Fanuc TP program (LS listing): UP002.LS

/PROG  UP002
/ATTR
OWNER		= AUROM;
COMMENT		= "Soldadura Est.";
PROG_SIZE	= 20204;
CREATE		= DATE 23-02-08  TIME 21:26:18;
MODIFIED	= DATE 24-04-03  TIME 04:58:58;
FILE_NAME	= UP002;
VERSION		= 0;
LINE_COUNT	= 81;
MEMORY_SIZE	= 39340;
PROTECT		= READ_WRITE;
TCD:  STACK_SIZE	= 500,
      TASK_PRIORITY	= 50,
      TIME_SLICE	= 0,
      BUSY_LAMP_OFF	= 0,
      ABORT_REQUEST	= 0,
      PAUSE_REQUEST	= 0;
DEFAULT_GROUP	= 1,1,1,1,*;
CONTROL_CODE	= 00000001 00000000;
/APPL
/MN
   1:  UFRAME_NUM=1 ;
   2:  UTOOL_NUM=2 ;
   3:  PAYLOAD[2] ;
   4:J P[1] 100% CNT0 ACC100 TB    .10sec,P-SPS    ;
      1:  TC_ONLINE (ON) ;
      2:  DO[23]=OFF ;
      3:  TIMER[4]=RESET ;
      4:  TIMER[4]=START ;
      5:  CALL MAKRO050    ;
      6:  !Lib. de Herramientas ;
      7:  DO[80]=ON ;
      8:  DO[78]=OFF ;
      9:  DO[77]=ON ;
     10:  DO[75]=OFF ;
     11:  !Lib. de Anticolisiones ;
     12:  DO[45]=ON ;
     13:  DO[46]=ON ;
     14:  !Apagar Posicion Base ;
     15:  DO[15]=OFF ;
     16:  !Roboter auf der Bahn ;
     17:  DO[16]=ON ;
     18:  !Basculante 1 en Pos. de Reposo ;
     19:  IF (!DI[842] AND DO[12]),CALL MAKRO072 ;
     20:  WAIT (M[96])    ;
     21:  WAIT (DI[23])    ;
     22:  DO[23]=(ON) ;
     23:  TC_ONLINE (M[1] AND M[30] AND M[32] AND M[33] AND M[95] AND M[96]) ;
       ------ ;
   5:J P[2] 100% CNT100 ACC100 TB   0.00sec,P-SPS    ;
      1:  TC_ONLINE (M[1] AND M[30] AND M[32] AND M[33] AND M[95] AND M[96]) ;
       ------ ;
   6:J P[3] 100% CNT100 ACC100 TB   0.00sec,P-SPS    ;
      1:  TC_ONLINE (M[1] AND M[30] AND M[32] AND M[33] AND M[95] AND M[96]) ;
       ------ ;
   7:J P[4] 100% CNT100 ACC100 TB   0.00sec,P-SPS    ;
      1:  TC_ONLINE (M[1] AND M[30] AND M[32] AND M[33] AND M[95] AND M[96]) ;
       ------ ;
   8:J P[5] 100% CNT90 ACC80 TB   0.00sec,P-SPS    ;
      1:  TC_ONLINE (M[1] AND M[30] AND M[32] AND M[33] AND M[95] AND M[96]) ;
       ------ ;
   9:  !5QA802035_014_O_PS_0007 ;
  10:  !Punto de Sol. No. 5737 ;
  11:J P[6] 100% CNT10 ACC80 TB    .10sec,P-SPS Offset,PR[11]    ;
      1:  TC_ONLINE (ON) ;
      2:  DO[23]=OFF ;
      3:  WAIT (!DI[16] AND DI[23])    ;
      4:  CALL VW_USER(Basic1,EZSP,Nr1,ProgNr=99, , ,S-Punkt=5737,Fzg_Typ=3,EIN/AUS=ON) ;
      5:  GO[2]=(R[197]) ;
      6:  WAIT (!DI[129] OR DI[26])    ;
      7:  CALL MAKRO080    ;
      8:  WAIT (DI[23])    ;
      9:  DO[23]=ON ;
     10:  TC_ONLINE (M[1] AND M[30] AND M[32] AND M[33] AND M[95] AND M[96]) ;
       ------ ;
  12:  !5QA802035_014_O_PS_0008 ;
  13:  !Punto de Sol. No. 5738 ;
  14:J P[7] 100% CNT0 ACC100 TB    .10sec,P-SPS Offset,PR[11]    ;
      1:  TC_ONLINE (ON) ;
      2:  DO[23]=OFF ;
      3:  WAIT (!DI[16] AND DI[23])    ;
      4:  CALL VW_USER(Basic1,EZSP,Nr1,ProgNr=99, , ,S-Punkt=5738,Fzg_Typ=3,EIN/AUS=ON) ;
      5:  GO[2]=(R[197]) ;
      6:  WAIT (!DI[129] OR DI[26])    ;
      7:  CALL MAKRO080    ;
      8:  WAIT (DI[23])    ;
      9:  DO[23]=ON ;
     10:  TC_ONLINE (M[1] AND M[30] AND M[32] AND M[33] AND M[95] AND M[96]) ;
       ------ ;
  15:  !5QA802035_014_O_PS_0009 ;
  16:  !Punto de Sol. No. 5739 ;
  17:J P[8] 100% CNT0 ACC100 TB    .10sec,P-SPS Offset,PR[11]    ;
      1:  TC_ONLINE (ON) ;
      2:  DO[23]=OFF ;
      3:  WAIT (!DI[16] AND DI[23])    ;
      4:  CALL VW_USER(Basic1,EZSP,Nr1,ProgNr=99, , ,S-Punkt=5739,Fzg_Typ=3,EIN/AUS=ON) ;
      5:  GO[2]=(R[197]) ;
      6:  WAIT (!DI[129] OR DI[26])    ;
      7:  CALL MAKRO080    ;
      8:  WAIT (DI[23])    ;
      9:  DO[23]=ON ;
     10:  TC_ONLINE (M[1] AND M[30] AND M[32] AND M[33] AND M[95] AND M[96]) ;
       ------ ;
  18:  !5QA802035_030_AE_PS_0004 ;
  19:  !Punto de Sol. No. 5740 ;
  20:J P[9] 100% CNT0 ACC100 TB    .10sec,P-SPS Offset,PR[11]    ;
      1:  TC_ONLINE (ON) ;
      2:  DO[23]=OFF ;
      3:  WAIT (!DI[16] AND DI[23])    ;
      4:  CALL VW_USER(Basic1,EZSP,Nr1,ProgNr=99, , ,S-Punkt=5740,Fzg_Typ=3,EIN/AUS=ON) ;
      5:  GO[2]=(R[197]) ;
      6:  WAIT (!DI[129] OR DI[26])    ;
      7:  CALL MAKRO080    ;
      8:  WAIT (DI[23])    ;
      9:  DO[23]=ON ;
     10:  TC_ONLINE (M[1] AND M[30] AND M[32] AND M[33] AND M[95] AND M[96]) ;
       ------ ;
  21:  !5QA802035_030_AE_PS_0005 ;
  22:  !Punto de Sol. No. 5741 ;
  23:J P[10] 100% CNT0 ACC100 TB    .10sec,P-SPS Offset,PR[11]    ;
      1:  TC_ONLINE (ON) ;
      2:  DO[23]=OFF ;
      3:  WAIT (!DI[16] AND DI[23])    ;
      4:  CALL VW_USER(Basic1,EZSP,Nr1,ProgNr=99, , ,S-Punkt=5741,Fzg_Typ=3,EIN/AUS=ON) ;
      5:  GO[2]=(R[197]) ;
      6:  WAIT (!DI[129] OR DI[26])    ;
      7:  CALL MAKRO080    ;
      8:  WAIT (DI[23])    ;
      9:  DO[23]=ON ;
     10:  TC_ONLINE (M[1] AND M[30] AND M[32] AND M[33] AND M[95] AND M[96]) ;
       ------ ;
  24:J P[11] 100% CNT100 ACC100 TB   0.00sec,P-SPS    ;
      1:  TC_ONLINE (M[1] AND M[30] AND M[32] AND M[33] AND M[95] AND M[96]) ;
       ------ ;
  25:  !5QA802035_030_AE_PS_0006 ;
  26:  !Punto de Sol. No. 5742 ;
  27:J P[12] 100% CNT0 ACC100 TB    .10sec,P-SPS Offset,PR[11]    ;
      1:  TC_ONLINE (ON) ;
      2:  DO[23]=OFF ;
      3:  WAIT (!DI[16] AND DI[23])    ;
      4:  CALL VW_USER(Basic1,EZSP,Nr1,ProgNr=99, , ,S-Punkt=5742,Fzg_Typ=3,EIN/AUS=ON) ;
      5:  GO[2]=(R[197]) ;
      6:  WAIT (!DI[129] OR DI[26])    ;
      7:  CALL MAKRO080    ;
      8:  WAIT (DI[23])    ;
      9:  DO[23]=ON ;
     10:  TC_ONLINE (M[1] AND M[30] AND M[32] AND M[33] AND M[95] AND M[96]) ;
       ------ ;
  28:J P[13] 100% CNT100 ACC100 TB   0.00sec,P-SPS    ;
      1:  TC_ONLINE (M[1] AND M[30] AND M[32] AND M[33] AND M[95] AND M[96]) ;
       ------ ;
  29:J P[14] 100% CNT100 ACC100 TB    .10sec,P-SPS    ;
      1:  TC_ONLINE (M[1] AND M[30] AND M[32] AND M[33] AND M[95] AND M[96]) ;
       ------ ;
  30:  !5QA802035_034_AJ_PS_0001 ;
  31:  !Punto de Sol. No. 5743 ;
  32:J P[15] 100% CNT0 ACC100 TB    .10sec,P-SPS Offset,PR[11]    ;
      1:  TC_ONLINE (ON) ;
      2:  DO[23]=OFF ;
      3:  WAIT (!DI[16] AND DI[23])    ;
      4:  CALL VW_USER(Basic1,EZSP,Nr1,ProgNr=99, , ,S-Punkt=5743,Fzg_Typ=3,EIN/AUS=ON) ;
      5:  GO[2]=(R[197]) ;
      6:  WAIT (!DI[129] OR DI[26])    ;
      7:  CALL MAKRO080    ;
      8:  WAIT (DI[23])    ;
      9:  DO[23]=ON ;
     10:  TC_ONLINE (M[1] AND M[30] AND M[32] AND M[33] AND M[95] AND M[96]) ;
       ------ ;
  33:  !5QA802035_034_AJ_PS_0003 ;
  34:  !Punto de Sol. No. 5744 ;
  35:J P[16] 100% CNT0 ACC100 TB    .10sec,P-SPS Offset,PR[11]    ;
      1:  TC_ONLINE (ON) ;
      2:  DO[23]=OFF ;
      3:  WAIT (!DI[16] AND DI[23])    ;
      4:  CALL VW_USER(Basic1,EZSP,Nr1,ProgNr=99, , ,S-Punkt=5744,Fzg_Typ=3,EIN/AUS=ON) ;
      5:  GO[2]=(R[197]) ;
      6:  WAIT (!DI[129] OR DI[26])    ;
      7:  CALL MAKRO080    ;
      8:  WAIT (DI[23])    ;
      9:  DO[23]=ON ;
     10:  TC_ONLINE (M[1] AND M[30] AND M[32] AND M[33] AND M[95] AND M[96]) ;
       ------ ;
  36:J P[17] 100% CNT100 ACC100 TB   0.00sec,P-SPS    ;
      1:  TC_ONLINE (M[1] AND M[30] AND M[32] AND M[33] AND M[95] AND M[96]) ;
       ------ ;
  37:J P[18] 100% CNT100 ACC100 TB   0.00sec,P-SPS    ;
      1:  TC_ONLINE (M[1] AND M[30] AND M[32] AND M[33] AND M[95] AND M[96]) ;
       ------ ;
  38:  !5QA802035_048_BL_PS_0001 ;
  39:  !Punto de Sol. No. 5749 ;
  40:J P[19] 100% CNT0 ACC100 TB    .10sec,P-SPS Offset,PR[11]    ;
      1:  TC_ONLINE (ON) ;
      2:  DO[23]=OFF ;
      3:  WAIT (!DI[16] AND DI[23])    ;
      4:  CALL VW_USER(Basic1,EZSP,Nr1,ProgNr=99, , ,S-Punkt=5749,Fzg_Typ=3,EIN/AUS=ON) ;
      5:  GO[2]=(R[197]) ;
      6:  WAIT (!DI[129] OR DI[26])    ;
      7:  CALL MAKRO080    ;
      8:  WAIT (DI[23])    ;
      9:  DO[23]=ON ;
     10:  TC_ONLINE (M[1] AND M[30] AND M[32] AND M[33] AND M[95] AND M[96]) ;
       ------ ;
  41:J P[20] 100% CNT100 ACC100 TB   0.00sec,P-SPS    ;
      1:  TC_ONLINE (M[1] AND M[30] AND M[32] AND M[33] AND M[95] AND M[96]) ;
       ------ ;
  42:J P[21] 100% CNT100 ACC100 TB   0.00sec,P-SPS    ;
      1:  TC_ONLINE (M[1] AND M[30] AND M[32] AND M[33] AND M[95] AND M[96]) ;
       ------ ;
  43:J P[22] 100% CNT100 ACC100 TB   0.00sec,P-SPS    ;
      1:  TC_ONLINE (M[1] AND M[30] AND M[32] AND M[33] AND M[95] AND M[96]) ;
       ------ ;
  44:J P[23] 100% CNT100 ACC100 TB   0.00sec,P-SPS    ;
      1:  TC_ONLINE (M[1] AND M[30] AND M[32] AND M[33] AND M[95] AND M[96]) ;
       ------ ;
  45:J P[24] 100% CNT100 ACC100 TB   0.00sec,P-SPS    ;
      1:  TC_ONLINE (M[1] AND M[30] AND M[32] AND M[33] AND M[95] AND M[96]) ;
       ------ ;
  46:J P[25] 100% CNT100 ACC100 TB   0.00sec,P-SPS    ;
      1:  TC_ONLINE (M[1] AND M[30] AND M[32] AND M[33] AND M[95] AND M[96]) ;
       ------ ;
  47:J P[26] 100% CNT100 ACC100 TB   0.00sec,P-SPS    ;
      1:  TC_ONLINE (M[1] AND M[30] AND M[32] AND M[33] AND M[95] AND M[96]) ;
       ------ ;
  48:J P[27] 100% CNT100 ACC100 TB   0.00sec,P-SPS    ;
      1:  TC_ONLINE (M[1] AND M[30] AND M[32] AND M[33] AND M[95] AND M[96]) ;
       ------ ;
  49:J P[28] 100% CNT100 ACC100 TB   0.00sec,P-SPS    ;
      1:  TC_ONLINE (M[1] AND M[30] AND M[32] AND M[33] AND M[95] AND M[96]) ;
       ------ ;
  50:J P[29] 100% CNT100 ACC100 TB   0.00sec,P-SPS    ;
      1:  TC_ONLINE (M[1] AND M[30] AND M[32] AND M[33] AND M[95] AND M[96]) ;
       ------ ;
  51:J P[30] 100% CNT100 ACC100 TB   0.00sec,P-SPS    ;
      1:  TC_ONLINE (M[1] AND M[30] AND M[32] AND M[33] AND M[95] AND M[96]) ;
       ------ ;
  52:J P[31] 100% CNT100 ACC100 TB   0.00sec,P-SPS    ;
      1:  TC_ONLINE (M[1] AND M[30] AND M[32] AND M[33] AND M[95] AND M[96]) ;
       ------ ;
  53:J P[32] 100% CNT100 ACC100 TB   0.00sec,P-SPS    ;
      1:  TC_ONLINE (M[1] AND M[30] AND M[32] AND M[33] AND M[95] AND M[96]) ;
       ------ ;
  54:  !5QA802035_042_AR_PS_0004 ;
  55:  !Punto de Sol. No. 5748 ;
  56:J P[33] 100% CNT0 ACC100 TB    .10sec,P-SPS Offset,PR[11]    ;
      1:  TC_ONLINE (ON) ;
      2:  DO[23]=OFF ;
      3:  WAIT (!DI[16] AND DI[23])    ;
      4:  CALL VW_USER(Basic1,EZSP,Nr1,ProgNr=99, , ,S-Punkt=5748,Fzg_Typ=3,EIN/AUS=ON) ;
      5:  GO[2]=(R[197]) ;
      6:  WAIT (!DI[129] OR DI[26])    ;
      7:  CALL MAKRO080    ;
      8:  WAIT (DI[23])    ;
      9:  DO[23]=ON ;
     10:  TC_ONLINE (M[1] AND M[30] AND M[32] AND M[33] AND M[95] AND M[96]) ;
       ------ ;
  57:  !5QA802035_042_AR_PS_0003 ;
  58:  !Punto de Sol. No. 5747 ;
  59:J P[34] 100% CNT0 ACC100 TB    .10sec,P-SPS Offset,PR[11]    ;
      1:  TC_ONLINE (ON) ;
      2:  DO[23]=OFF ;
      3:  WAIT (!DI[16] AND DI[23])    ;
      4:  CALL VW_USER(Basic1,EZSP,Nr1,ProgNr=99, , ,S-Punkt=5747,Fzg_Typ=3,EIN/AUS=ON) ;
      5:  GO[2]=(R[197]) ;
      6:  WAIT (!DI[129] OR DI[26])    ;
      7:  CALL MAKRO080    ;
      8:  WAIT (DI[23])    ;
      9:  DO[23]=ON ;
     10:  TC_ONLINE (M[1] AND M[30] AND M[32] AND M[33] AND M[95] AND M[96]) ;
       ------ ;
  60:J P[35] 100% CNT100 ACC100 TB   0.00sec,P-SPS    ;
      1:  TC_ONLINE (M[1] AND M[30] AND M[32] AND M[33] AND M[95] AND M[96]) ;
       ------ ;
  61:J P[36] 100% CNT100 ACC100 TB   0.00sec,P-SPS    ;
      1:  TC_ONLINE (M[1] AND M[30] AND M[32] AND M[33] AND M[95] AND M[96]) ;
       ------ ;
  62:J P[37] 100% CNT100 ACC100 TB   0.00sec,P-SPS    ;
      1:  TC_ONLINE (M[1] AND M[30] AND M[32] AND M[33] AND M[95] AND M[96]) ;
       ------ ;
  63:J P[38] 100% CNT100 ACC100 TB   0.00sec,P-SPS    ;
      1:  TC_ONLINE (M[1] AND M[30] AND M[32] AND M[33] AND M[95] AND M[96]) ;
       ------ ;
  64:J P[39] 100% CNT100 ACC100 TB   0.00sec,P-SPS    ;
      1:  TC_ONLINE (M[1] AND M[30] AND M[32] AND M[33] AND M[95] AND M[96]) ;
       ------ ;
  65:J P[40] 100% CNT100 ACC100 TB   0.00sec,P-SPS    ;
      1:  TC_ONLINE (M[1] AND M[30] AND M[32] AND M[33] AND M[95] AND M[96]) ;
       ------ ;
  66:J P[41] 100% CNT100 ACC100 TB   0.00sec,P-SPS    ;
      1:  TC_ONLINE (M[1] AND M[30] AND M[32] AND M[33] AND M[95] AND M[96]) ;
       ------ ;
  67:J P[42] 100% CNT0 ACC100 TB   0.00sec,P-SPS    ;
      1:  TC_ONLINE (M[1] AND M[30] AND M[32] AND M[33] AND M[95] AND M[96]) ;
       ------ ;
  68:  !5QA802035_042_AR_PS_0001 ;
  69:  !Punto de Sol. No. 5745 ;
  70:J P[43] 100% CNT0 ACC100 TB    .10sec,P-SPS Offset,PR[11]    ;
      1:  TC_ONLINE (ON) ;
      2:  DO[23]=OFF ;
      3:  WAIT (!DI[16] AND DI[23])    ;
      4:  CALL VW_USER(Basic1,EZSP,Nr1,ProgNr=99, , ,S-Punkt=5745,Fzg_Typ=3,EIN/AUS=ON) ;
      5:  GO[2]=(R[197]-5) ;
      6:  WAIT (!DI[129] OR DI[26])    ;
      7:  CALL MAKRO080    ;
      8:  WAIT (DI[23])    ;
      9:  DO[23]=ON ;
     10:  TC_ONLINE (M[1] AND M[30] AND M[32] AND M[33] AND M[95] AND M[96]) ;
       ------ ;
  71:  !5QA802035_042_AR_PS_0002 ;
  72:  !Punto de Sol. No. 5746 ;
  73:  !Fin de Trabajo 2 ;
  74:J P[44] 100% CNT0 ACC100 TB    .10sec,P-SPS Offset,PR[11]    ;
      1:  TC_ONLINE (ON) ;
      2:  DO[23]=OFF ;
      3:  WAIT (!DI[16] AND DI[23])    ;
      4:  CALL VW_USER(Basic1,EZSP,Nr1,ProgNr=99, , ,S-Punkt=5746,Fzg_Typ=3,EIN/AUS=ON) ;
      5:  GO[2]=(R[197]) ;
      6:  WAIT (!DI[129] OR DI[26])    ;
      7:  CALL MAKRO080    ;
      8:  IF (!DI[145] AND !DI[129]),CALL MAKRO002 ;
      9:  WAIT (DI[23])    ;
     10:  DO[23]=ON ;
     11:  TC_ONLINE (M[1] AND M[30] AND M[32] AND M[33] AND M[95] AND M[96]) ;
       ------ ;
  75:J P[45] 100% CNT100 ACC100 TB   0.00sec,P-SPS    ;
      1:  TC_ONLINE (M[1] AND M[30] AND M[32] AND M[33] AND M[95] AND M[96]) ;
       ------ ;
  76:J P[46] 100% CNT100 ACC100 TB   0.00sec,P-SPS    ;
      1:  TC_ONLINE (M[1] AND M[30] AND M[32] AND M[33] AND M[95] AND M[96]) ;
       ------ ;
  77:J P[47] 100% CNT100 ACC100 TB   0.00sec,P-SPS    ;
      1:  TC_ONLINE (M[1] AND M[30] AND M[32] AND M[33] AND M[95] AND M[96]) ;
       ------ ;
  78:J P[48] 100% CNT100 ACC100 TB   0.00sec,P-SPS    ;
      1:  TC_ONLINE (M[1] AND M[30] AND M[32] AND M[33] AND M[95] AND M[96]) ;
       ------ ;
  79:J P[49] 100% CNT100 ACC100 TB   0.00sec,P-SPS    ;
      1:  TC_ONLINE (M[1] AND M[30] AND M[32] AND M[33] AND M[95] AND M[96]) ;
       ------ ;
  80:J P[50] 100% CNT100 ACC100 TB   0.00sec,P-SPS    ;
      1:  TC_ONLINE (M[1] AND M[30] AND M[32] AND M[33] AND M[95] AND M[96]) ;
       ------ ;
  81:J P[51] 100% CNT0 ACC100 TB    .10sec,P-SPS    ;
      1:  TC_ONLINE (ON) ;
      2:  DO[23]=OFF ;
      3:  TIMER[4]=STOP ;
      4:  CALL VW_USER(Basic1,EZSP,Nr1,ProgNr=31, , ,S-Punkt=31, ,EIN/AUS=1) ;
      5:  WAIT (DI[23])    ;
      6:  DO[23]=ON ;
      7:  TC_ONLINE (M[1] AND M[30] AND M[32] AND M[33] AND M[95] AND M[96]) ;
       ------ ;
/POS
P[1]{
   GP1:
	UF : 1, UT : 2,		CONFIG : 'N U T, 0, 0, 0',
	RX = -1944.900  mm,	RY =  1526.189  mm,	RZ =  -496.255  mm,
	RW =    55.263 deg,	RP =     4.579 deg,	RR =  -173.433 deg
   GP2:
	UF : 1, UT : 2,
	J1=   100.000  mm
   GP3:
	UF : 1, UT : 2,
	J1=     0.000  mm
   GP4:
	UF : 1, UT : 2,
	J1=     0.000  mm
};
P[2]{
   GP1:
	UF : 1, UT : 2,		CONFIG : 'N U T, 0, 0, 0',
	RX =   179.234  mm,	RY =   151.690  mm,	RZ =  -253.733  mm,
	RW =   135.376 deg,	RP =    18.701 deg,	RR =   -99.313 deg
   GP2:
	UF : 1, UT : 2,
	J1=    82.425  mm
   GP3:
	UF : 1, UT : 2,
	J1=     0.000  mm
   GP4:
	UF : 1, UT : 2,
	J1=     0.000  mm
};
P[3]{
   GP1:
	UF : 1, UT : 2,		CONFIG : 'N U T, 0, 0, 0',
	RX =   308.340  mm,	RY =   144.764  mm,	RZ =    90.903  mm,
	RW =   144.538 deg,	RP =    12.921 deg,	RR =   -94.764 deg
   GP2:
	UF : 1, UT : 2,
	J1=    83.242  mm
   GP3:
	UF : 1, UT : 2,
	J1=     0.000  mm
   GP4:
	UF : 1, UT : 2,
	J1=     0.000  mm
};
P[4]{
   GP1:
	UF : 1, UT : 2,		CONFIG : 'N U T, 0, 0, 0',
	RX =   290.098  mm,	RY =   377.472  mm,	RZ =    85.805  mm,
	RW =   146.739 deg,	RP =     7.916 deg,	RR =   -94.914 deg
   GP2:
	UF : 1, UT : 2,
	J1=    70.000  mm
   GP3:
	UF : 1, UT : 2,
	J1=     0.000  mm
   GP4:
	UF : 1, UT : 2,
	J1=     0.000  mm
};
P[5]{
   GP1:
	UF : 1, UT : 2,		CONFIG : 'N U T, 0, 0, 0',
	RX =   248.363  mm,	RY =   385.106  mm,	RZ =    32.759  mm,
	RW =   141.741 deg,	RP =     7.911 deg,	RR =   -94.917 deg
   GP2:
	UF : 1, UT : 2,
	J1=   107.800  mm
   GP3:
	UF : 1, UT : 2,
	J1=     0.000  mm
   GP4:
	UF : 1, UT : 2,
	J1=     0.000  mm
};
P[6]{
   GP1:
	UF : 1, UT : 2,		CONFIG : 'N U T, 0, 0, 0',
	RX =   186.578  mm,	RY =   385.883  mm,	RZ =    37.075  mm,
	RW =   141.518 deg,	RP =     8.520 deg,	RR =   -96.184 deg
   GP2:
	UF : 1, UT : 2,
	J1=    27.000  mm
   GP3:
	UF : 1, UT : 2,
	J1=     0.000  mm
   GP4:
	UF : 1, UT : 2,
	J1=     0.000  mm
};
P[7]{
   GP1:
	UF : 1, UT : 2,		CONFIG : 'N U T, 0, 0, 0',
	RX =   183.514  mm,	RY =   380.431  mm,	RZ =    20.676  mm,
	RW =   142.050 deg,	RP =     8.705 deg,	RR =   -96.668 deg
   GP2:
	UF : 1, UT : 2,
	J1=    22.000  mm
   GP3:
	UF : 1, UT : 2,
	J1=     0.000  mm
   GP4:
	UF : 1, UT : 2,
	J1=     0.000  mm
};
P[8]{
   GP1:
	UF : 1, UT : 2,		CONFIG : 'N U T, 0, 0, 0',
	RX =   176.359  mm,	RY =   387.068  mm,	RZ =    33.122  mm,
	RW =   141.586 deg,	RP =     8.467 deg,	RR =   -99.117 deg
   GP2:
	UF : 1, UT : 2,
	J1=    24.600  mm
   GP3:
	UF : 1, UT : 2,
	J1=     0.000  mm
   GP4:
	UF : 1, UT : 2,
	J1=     0.000  mm
};
P[9]{
   GP1:
	UF : 1, UT : 2,		CONFIG : 'N U T, 0, 0, 0',
	RX =   152.752  mm,	RY =   386.059  mm,	RZ =    46.973  mm,
	RW =   144.004 deg,	RP =     7.570 deg,	RR =   -97.106 deg
   GP2:
	UF : 1, UT : 2,
	J1=    25.000  mm
   GP3:
	UF : 1, UT : 2,
	J1=     0.000  mm
   GP4:
	UF : 1, UT : 2,
	J1=     0.000  mm
};
P[10]{
   GP1:
	UF : 1, UT : 2,		CONFIG : 'N U T, 0, 0, 0',
	RX =   148.722  mm,	RY =   380.556  mm,	RZ =    64.424  mm,
	RW =   142.523 deg,	RP =     9.712 deg,	RR =   -94.121 deg
   GP2:
	UF : 1, UT : 2,
	J1=    19.800  mm
   GP3:
	UF : 1, UT : 2,
	J1=     0.000  mm
   GP4:
	UF : 1, UT : 2,
	J1=     0.000  mm
};
P[11]{
   GP1:
	UF : 1, UT : 2,		CONFIG : 'N U T, 0, 0, 0',
	RX =   128.750  mm,	RY =   386.943  mm,	RZ =    69.419  mm,
	RW =   130.513 deg,	RP =     7.592 deg,	RR =   -95.471 deg
   GP2:
	UF : 1, UT : 2,
	J1=    17.508  mm
   GP3:
	UF : 1, UT : 2,
	J1=     0.000  mm
   GP4:
	UF : 1, UT : 2,
	J1=     0.000  mm
};
P[12]{
   GP1:
	UF : 1, UT : 2,		CONFIG : 'N U T, 0, 0, 0',
	RX =   126.104  mm,	RY =   385.644  mm,	RZ =    63.431  mm,
	RW =   123.356 deg,	RP =     7.161 deg,	RR =   -97.236 deg
   GP2:
	UF : 1, UT : 2,
	J1=    25.000  mm
   GP3:
	UF : 1, UT : 2,
	J1=     0.000  mm
   GP4:
	UF : 1, UT : 2,
	J1=     0.000  mm
};
P[13]{
   GP1:
	UF : 1, UT : 2,		CONFIG : 'N U T, 0, 0, 0',
	RX =   118.622  mm,	RY =   388.682  mm,	RZ =    80.415  mm,
	RW =   120.718 deg,	RP =     6.449 deg,	RR =   -96.850 deg
   GP2:
	UF : 1, UT : 2,
	J1=    70.000  mm
   GP3:
	UF : 1, UT : 2,
	J1=     0.000  mm
   GP4:
	UF : 1, UT : 2,
	J1=     0.000  mm
};
P[14]{
   GP1:
	UF : 1, UT : 2,		CONFIG : 'N U T, 0, 0, 0',
	RX =   118.638  mm,	RY =   386.921  mm,	RZ =   128.143  mm,
	RW =   108.283 deg,	RP =     5.033 deg,	RR =  -100.823 deg
   GP2:
	UF : 1, UT : 2,
	J1=    70.000  mm
   GP3:
	UF : 1, UT : 2,
	J1=     0.000  mm
   GP4:
	UF : 1, UT : 2,
	J1=     0.000  mm
};
P[15]{
   GP1:
	UF : 1, UT : 2,		CONFIG : 'N U T, 0, 0, 0',
	RX =   120.000  mm,	RY =   378.399  mm,	RZ =   125.152  mm,
	RW =   108.102 deg,	RP =     -.004 deg,	RR =  -102.385 deg
   GP2:
	UF : 1, UT : 2,
	J1=    22.400  mm
   GP3:
	UF : 1, UT : 2,
	J1=     0.000  mm
   GP4:
	UF : 1, UT : 2,
	J1=     0.000  mm
};
P[16]{
   GP1:
	UF : 1, UT : 2,		CONFIG : 'N U T, 0, 0, 0',
	RX =   132.327  mm,	RY =   376.009  mm,	RZ =   125.928  mm,
	RW =   102.710 deg,	RP =     2.034 deg,	RR =  -100.568 deg
   GP2:
	UF : 1, UT : 2,
	J1=    22.100  mm
   GP3:
	UF : 1, UT : 2,
	J1=     0.000  mm
   GP4:
	UF : 1, UT : 2,
	J1=     0.000  mm
};
P[17]{
   GP1:
	UF : 1, UT : 2,		CONFIG : 'N U T, 0, 0, 0',
	RX =   131.372  mm,	RY =   383.685  mm,	RZ =   128.549  mm,
	RW =   102.732 deg,	RP =     6.408 deg,	RR =   -99.926 deg
   GP2:
	UF : 1, UT : 2,
	J1=    80.000  mm
   GP3:
	UF : 1, UT : 2,
	J1=     0.000  mm
   GP4:
	UF : 1, UT : 2,
	J1=     0.000  mm
};
P[18]{
   GP1:
	UF : 1, UT : 2,		CONFIG : 'N U T, 0, 0, 0',
	RX =   155.761  mm,	RY =   375.193  mm,	RZ =   151.816  mm,
	RW =    89.691 deg,	RP =     2.702 deg,	RR =   -96.536 deg
   GP2:
	UF : 1, UT : 2,
	J1=    80.000  mm
   GP3:
	UF : 1, UT : 2,
	J1=     0.000  mm
   GP4:
	UF : 1, UT : 2,
	J1=     0.000  mm
};
P[19]{
   GP1:
	UF : 1, UT : 2,		CONFIG : 'N U T, 0, 0, 0',
	RX =   158.529  mm,	RY =   367.613  mm,	RZ =   154.919  mm,
	RW =    89.801 deg,	RP =     -.458 deg,	RR =   -99.347 deg
   GP2:
	UF : 1, UT : 2,
	J1=    10.600  mm
   GP3:
	UF : 1, UT : 2,
	J1=     0.000  mm
   GP4:
	UF : 1, UT : 2,
	J1=     0.000  mm
};
P[20]{
   GP1:
	UF : 1, UT : 2,		CONFIG : 'N U T, 0, 0, 0',
	RX =   155.761  mm,	RY =   375.193  mm,	RZ =   151.816  mm,
	RW =    89.691 deg,	RP =     2.702 deg,	RR =   -96.536 deg
   GP2:
	UF : 1, UT : 2,
	J1=    80.000  mm
   GP3:
	UF : 1, UT : 2,
	J1=     0.000  mm
   GP4:
	UF : 1, UT : 2,
	J1=     0.000  mm
};
P[21]{
   GP1:
	UF : 1, UT : 2,		CONFIG : 'N U T, 0, 0, 0',
	RX =   131.372  mm,	RY =   383.685  mm,	RZ =   128.549  mm,
	RW =   102.732 deg,	RP =     6.408 deg,	RR =   -99.926 deg
   GP2:
	UF : 1, UT : 2,
	J1=    80.000  mm
   GP3:
	UF : 1, UT : 2,
	J1=     0.000  mm
   GP4:
	UF : 1, UT : 2,
	J1=     0.000  mm
};
P[22]{
   GP1:
	UF : 1, UT : 2,		CONFIG : 'N U T, 0, 0, 0',
	RX =   133.597  mm,	RY =   390.864  mm,	RZ =    69.630  mm,
	RW =   115.740 deg,	RP =     7.913 deg,	RR =   -94.913 deg
   GP2:
	UF : 1, UT : 2,
	J1=   100.000  mm
   GP3:
	UF : 1, UT : 2,
	J1=     0.000  mm
   GP4:
	UF : 1, UT : 2,
	J1=     0.000  mm
};
P[23]{
   GP1:
	UF : 1, UT : 2,		CONFIG : 'N U T, 0, 0, 0',
	RX =   235.695  mm,	RY =   386.669  mm,	RZ =    31.528  mm,
	RW =   132.739 deg,	RP =     7.916 deg,	RR =   -94.914 deg
   GP2:
	UF : 1, UT : 2,
	J1=   100.000  mm
   GP3:
	UF : 1, UT : 2,
	J1=     0.000  mm
   GP4:
	UF : 1, UT : 2,
	J1=     0.000  mm
};
P[24]{
   GP1:
	UF : 1, UT : 2,		CONFIG : 'N U T, 0, 0, 0',
	RX =   290.722  mm,	RY =   370.916  mm,	RZ =    86.736  mm,
	RW =   146.739 deg,	RP =     7.916 deg,	RR =   -94.914 deg
   GP2:
	UF : 1, UT : 2,
	J1=   100.000  mm
   GP3:
	UF : 1, UT : 2,
	J1=     0.000  mm
   GP4:
	UF : 1, UT : 2,
	J1=     0.000  mm
};
P[25]{
   GP1:
	UF : 1, UT : 2,		CONFIG : 'N U T, 0, 0, 0',
	RX =   271.679  mm,	RY =   148.864  mm,	RZ =    55.561  mm,
	RW =   141.740 deg,	RP =     7.915 deg,	RR =   -94.915 deg
   GP2:
	UF : 1, UT : 2,
	J1=   100.000  mm
   GP3:
	UF : 1, UT : 2,
	J1=     0.000  mm
   GP4:
	UF : 1, UT : 2,
	J1=     0.000  mm
};
P[26]{
   GP1:
	UF : 1, UT : 2,		CONFIG : 'N U T, 0, 0, 0',
	RX =   -19.391  mm,	RY =  -117.451  mm,	RZ =  -293.687  mm,
	RW =   128.511 deg,	RP =    27.818 deg,	RR =  -107.115 deg
   GP2:
	UF : 1, UT : 2,
	J1=   100.000  mm
   GP3:
	UF : 1, UT : 2,
	J1=     0.000  mm
   GP4:
	UF : 1, UT : 2,
	J1=     0.000  mm
};
P[27]{
   GP1:
	UF : 1, UT : 2,		CONFIG : 'N U T, 0, 0, 0',
	RX =  -497.400  mm,	RY =  -491.963  mm,	RZ =   113.189  mm,
	RW =    90.776 deg,	RP =    -2.355 deg,	RR =   -98.987 deg
   GP2:
	UF : 1, UT : 2,
	J1=   100.000  mm
   GP3:
	UF : 1, UT : 2,
	J1=     0.000  mm
   GP4:
	UF : 1, UT : 2,
	J1=     0.000  mm
};
P[28]{
   GP1:
	UF : 1, UT : 2,		CONFIG : 'F U T, 0, 0, 0',
	RX =  -672.602  mm,	RY =   376.473  mm,	RZ =  -233.136  mm,
	RW =    20.959 deg,	RP =    60.535 deg,	RR =  -135.996 deg
   GP2:
	UF : 1, UT : 2,
	J1=   100.000  mm
   GP3:
	UF : 1, UT : 2,
	J1=     0.000  mm
   GP4:
	UF : 1, UT : 2,
	J1=     0.000  mm
};
P[29]{
   GP1:
	UF : 1, UT : 2,		CONFIG : 'F U T, 0, 0, 0',
	RX =  -414.322  mm,	RY =   269.978  mm,	RZ =  -204.977  mm,
	RW =    22.192 deg,	RP =    69.151 deg,	RR =  -113.679 deg
   GP2:
	UF : 1, UT : 2,
	J1=   100.000  mm
   GP3:
	UF : 1, UT : 2,
	J1=     0.000  mm
   GP4:
	UF : 1, UT : 2,
	J1=     0.000  mm
};
P[30]{
   GP1:
	UF : 1, UT : 2,		CONFIG : 'F U T, 0, 0, 0',
	RX =  -138.424  mm,	RY =   567.302  mm,	RZ =  -128.526  mm,
	RW =   -93.054 deg,	RP =    88.166 deg,	RR =   176.944 deg
   GP2:
	UF : 1, UT : 2,
	J1=   100.000  mm
   GP3:
	UF : 1, UT : 2,
	J1=     0.000  mm
   GP4:
	UF : 1, UT : 2,
	J1=     0.000  mm
};
P[31]{
   GP1:
	UF : 1, UT : 2,		CONFIG : 'F U T, 0, 0, 0',
	RX =  -128.072  mm,	RY =   585.429  mm,	RZ =   194.048  mm,
	RW =   -93.052 deg,	RP =    88.166 deg,	RR =   176.947 deg
   GP2:
	UF : 1, UT : 2,
	J1=    65.000  mm
   GP3:
	UF : 1, UT : 2,
	J1=     0.000  mm
   GP4:
	UF : 1, UT : 2,
	J1=     0.000  mm
};
P[32]{
   GP1:
	UF : 1, UT : 2,		CONFIG : 'F U T, 0, 0, 0',
	RX =  -128.650  mm,	RY =   466.699  mm,	RZ =   175.021  mm,
	RW =   -93.051 deg,	RP =    88.166 deg,	RR =   176.948 deg
   GP2:
	UF : 1, UT : 2,
	J1=    65.000  mm
   GP3:
	UF : 1, UT : 2,
	J1=     0.000  mm
   GP4:
	UF : 1, UT : 2,
	J1=     0.000  mm
};
P[33]{
   GP1:
	UF : 1, UT : 2,		CONFIG : 'F U T, 0, 0, 0',
	RX =  -128.642  mm,	RY =   468.510  mm,	RZ =   164.022  mm,
	RW =  -172.224 deg,	RP =    87.133 deg,	RR =    97.808 deg
   GP2:
	UF : 1, UT : 2,
	J1=    29.000  mm
   GP3:
	UF : 1, UT : 2,
	J1=     0.000  mm
   GP4:
	UF : 1, UT : 2,
	J1=     0.000  mm
};
P[34]{
   GP1:
	UF : 1, UT : 2,		CONFIG : 'F U T, 0, 0, 0',
	RX =  -115.319  mm,	RY =   462.871  mm,	RZ =   164.314  mm,
	RW =  -150.201 deg,	RP =    86.018 deg,	RR =   119.740 deg
   GP2:
	UF : 1, UT : 2,
	J1=    29.000  mm
   GP3:
	UF : 1, UT : 2,
	J1=     0.000  mm
   GP4:
	UF : 1, UT : 2,
	J1=     0.000  mm
};
P[35]{
   GP1:
	UF : 1, UT : 2,		CONFIG : 'F U T, 0, 0, 0',
	RX =  -113.875  mm,	RY =   463.805  mm,	RZ =   170.331  mm,
	RW =   -90.130 deg,	RP =    86.342 deg,	RR =   179.870 deg
   GP2:
	UF : 1, UT : 2,
	J1=    65.000  mm
   GP3:
	UF : 1, UT : 2,
	J1=     0.000  mm
   GP4:
	UF : 1, UT : 2,
	J1=     0.000  mm
};
P[36]{
   GP1:
	UF : 1, UT : 2,		CONFIG : 'F U T, 0, 0, 0',
	RX =  -128.671  mm,	RY =   566.741  mm,	RZ =   175.305  mm,
	RW =   -93.052 deg,	RP =    88.166 deg,	RR =   176.947 deg
   GP2:
	UF : 1, UT : 2,
	J1=    65.000  mm
   GP3:
	UF : 1, UT : 2,
	J1=     0.000  mm
   GP4:
	UF : 1, UT : 2,
	J1=     0.000  mm
};
P[37]{
   GP1:
	UF : 1, UT : 2,		CONFIG : 'F U T, 0, 0, 0',
	RX =  -138.421  mm,	RY =   567.300  mm,	RZ =  -128.527  mm,
	RW =   -93.055 deg,	RP =    88.166 deg,	RR =   176.944 deg
   GP2:
	UF : 1, UT : 2,
	J1=   100.000  mm
   GP3:
	UF : 1, UT : 2,
	J1=     0.000  mm
   GP4:
	UF : 1, UT : 2,
	J1=     0.000  mm
};
P[38]{
   GP1:
	UF : 1, UT : 2,		CONFIG : 'F U T, 0, 0, 0',
	RX =   138.829  mm,	RY =   182.570  mm,	RZ =  -249.227  mm,
	RW =    -8.150 deg,	RP =    76.970 deg,	RR =    -7.943 deg
   GP2:
	UF : 1, UT : 2,
	J1=   100.000  mm
   GP3:
	UF : 1, UT : 2,
	J1=     0.000  mm
   GP4:
	UF : 1, UT : 2,
	J1=     0.000  mm
};
P[39]{
   GP1:
	UF : 1, UT : 2,		CONFIG : 'N U T, 0, 0, 0',
	RX =   231.483  mm,	RY =   842.822  mm,	RZ =  -247.302  mm,
	RW =    79.006 deg,	RP =    20.120 deg,	RR =    71.460 deg
   GP2:
	UF : 1, UT : 2,
	J1=   100.000  mm
   GP3:
	UF : 1, UT : 2,
	J1=     0.000  mm
   GP4:
	UF : 1, UT : 2,
	J1=     0.000  mm
};
P[40]{
   GP1:
	UF : 1, UT : 2,		CONFIG : 'N U T, 0, 0, 0',
	RX =    42.824  mm,	RY =   383.411  mm,	RZ =  -208.905  mm,
	RW =    53.051 deg,	RP =     9.546 deg,	RR =    66.707 deg
   GP2:
	UF : 1, UT : 2,
	J1=   100.000  mm
   GP3:
	UF : 1, UT : 2,
	J1=     0.000  mm
   GP4:
	UF : 1, UT : 2,
	J1=     0.000  mm
};
P[41]{
   GP1:
	UF : 1, UT : 2,		CONFIG : 'N U T, 0, 0, 0',
	RX =  -117.859  mm,	RY =   428.006  mm,	RZ =    35.475  mm,
	RW =    53.011 deg,	RP =     -.041 deg,	RR =    73.928 deg
   GP2:
	UF : 1, UT : 2,
	J1=   100.000  mm
   GP3:
	UF : 1, UT : 2,
	J1=     0.000  mm
   GP4:
	UF : 1, UT : 2,
	J1=     0.000  mm
};
P[42]{
   GP1:
	UF : 1, UT : 2,		CONFIG : 'N U T, 0, 0, 0',
	RX =  -116.157  mm,	RY =   433.764  mm,	RZ =   185.574  mm,
	RW =    53.011 deg,	RP =     -.040 deg,	RR =    73.926 deg
   GP2:
	UF : 1, UT : 2,
	J1=   100.000  mm
   GP3:
	UF : 1, UT : 2,
	J1=     0.000  mm
   GP4:
	UF : 1, UT : 2,
	J1=     0.000  mm
};
P[43]{
   GP1:
	UF : 1, UT : 2,		CONFIG : 'N U T, 0, 0, 0',
	RX =  -116.518  mm,	RY =   450.372  mm,	RZ =   183.473  mm,
	RW =    53.020 deg,	RP =     -.424 deg,	RR =    75.260 deg
   GP2:
	UF : 1, UT : 2,
	J1=    20.500  mm
   GP3:
	UF : 1, UT : 2,
	J1=     0.000  mm
   GP4:
	UF : 1, UT : 2,
	J1=     0.000  mm
};
P[44]{
   GP1:
	UF : 1, UT : 2,		CONFIG : 'N U T, 0, 0, 0',
	RX =  -133.232  mm,	RY =   449.602  mm,	RZ =   182.905  mm,
	RW =    52.965 deg,	RP =      .235 deg,	RR =    77.078 deg
   GP2:
	UF : 1, UT : 2,
	J1=    25.500  mm
   GP3:
	UF : 1, UT : 2,
	J1=     0.000  mm
   GP4:
	UF : 1, UT : 2,
	J1=     0.000  mm
};
P[45]{
   GP1:
	UF : 1, UT : 2,		CONFIG : 'N U T, 0, 0, 0',
	RX =  -132.206  mm,	RY =   438.002  mm,	RZ =   186.393  mm,
	RW =    52.980 deg,	RP =      .083 deg,	RR =    76.731 deg
   GP2:
	UF : 1, UT : 2,
	J1=   100.000  mm
   GP3:
	UF : 1, UT : 2,
	J1=     0.000  mm
   GP4:
	UF : 1, UT : 2,
	J1=     0.000  mm
};
P[46]{
   GP1:
	UF : 1, UT : 2,		CONFIG : 'N U T, 0, 0, 0',
	RX =  -100.324  mm,	RY =   416.245  mm,	RZ =   135.424  mm,
	RW =    52.980 deg,	RP =      .083 deg,	RR =    76.731 deg
   GP2:
	UF : 1, UT : 2,
	J1=   100.000  mm
   GP3:
	UF : 1, UT : 2,
	J1=     0.000  mm
   GP4:
	UF : 1, UT : 2,
	J1=     0.000  mm
};
P[47]{
   GP1:
	UF : 1, UT : 2,		CONFIG : 'N U T, 0, 0, 0',
	RX =   -95.539  mm,	RY =   401.367  mm,	RZ =    54.900  mm,
	RW =    52.993 deg,	RP =     2.775 deg,	RR =    76.212 deg
   GP2:
	UF : 1, UT : 2,
	J1=   100.000  mm
   GP3:
	UF : 1, UT : 2,
	J1=     0.000  mm
   GP4:
	UF : 1, UT : 2,
	J1=     0.000  mm
};
P[48]{
   GP1:
	UF : 1, UT : 2,		CONFIG : 'N U T, 0, 0, 0',
	RX =   109.401  mm,	RY =    24.179  mm,	RZ =  -204.626  mm,
	RW =    50.962 deg,	RP =    15.750 deg,	RR =    63.377 deg
   GP2:
	UF : 1, UT : 2,
	J1=   100.000  mm
   GP3:
	UF : 1, UT : 2,
	J1=     0.000  mm
   GP4:
	UF : 1, UT : 2,
	J1=     0.000  mm
};
P[49]{
   GP1:
	UF : 1, UT : 2,		CONFIG : 'N U T, 0, 0, 0',
	RX =  -722.148  mm,	RY =    43.278  mm,	RZ =  -327.065  mm,
	RW =    46.966 deg,	RP =    47.732 deg,	RR =   -42.290 deg
   GP2:
	UF : 1, UT : 2,
	J1=   100.000  mm
   GP3:
	UF : 1, UT : 2,
	J1=     0.000  mm
   GP4:
	UF : 1, UT : 2,
	J1=     0.000  mm
};
P[50]{
   GP1:
	UF : 1, UT : 2,		CONFIG : 'N U T, 0, 0, 0',
	RX =  -570.106  mm,	RY =   808.033  mm,	RZ = -1141.611  mm,
	RW =    65.605 deg,	RP =    37.828 deg,	RR =  -126.474 deg
   GP2:
	UF : 1, UT : 2,
	J1=   100.000  mm
   GP3:
	UF : 1, UT : 2,
	J1=     0.000  mm
   GP4:
	UF : 1, UT : 2,
	J1=     0.000  mm
};
P[51]{
   GP1:
	UF : 1, UT : 2,		CONFIG : 'N U T, 0, 0, 0',
	RX = -1944.900  mm,	RY =  1526.189  mm,	RZ =  -496.255  mm,
	RW =    55.263 deg,	RP =     4.579 deg,	RR =  -173.433 deg
   GP2:
	UF : 1, UT : 2,
	J1=   100.000  mm
   GP3:
	UF : 1, UT : 2,
	J1=     0.000  mm
   GP4:
	UF : 1, UT : 2,
	J1=     0.000  mm
};
/END
